(* IEC 61131-3 sources: TIA2AX/tests/test_projects/expected/HW_2200330_V18/ST30_PLC, 6 files *)

(* ---- HwInputs.st ---- *)
TYPE
	HwInputs : STRUCT
		ST30_ET200SP_CM_4xIO_Link_1 AT %B100 : ARRAY[0..31] OF BYTE;
		ST30_ET200SP_CM_4xIO_Link_2 AT %B132 : ARRAY[0..31] OF BYTE;
		ST30_ET200SP_DI_16x24VDC_ST_1 AT %B0 : WORD;
		ST30_ET200SP_DI_16x24VDC_ST_2 AT %B2 : WORD;
		ST30_ET200SP_DI_16x24VDC_ST_3 AT %B4 : WORD;
		ST30_ET200SP_DI_16x24VDC_ST_4 AT %B6 : WORD;
		ST30_ET200SP_DI_16x24VDC_ST_5 AT %B8 : WORD;
		ST30_ET200SP_DI_16x24VDC_ST_6 AT %B10 : WORD;
		ST30_1_DM260_Acquisition_Status_1 AT %B1500 : ARRAY[0..2] OF BYTE;
		ST30_1_DM260_Results_Status_1 AT %B1503 : BYTE;
		ST30_1_DM260_Soft_Event_Control_1 AT %B1504 : BYTE;
		ST30_1_DM260_Result_Data_64_bytes_1 AT %B1510 : ARRAY[0..71] OF BYTE;
		ST30_2_DM260_Acquisition_Status_1 AT %B2500 : ARRAY[0..2] OF BYTE;
		ST30_2_DM260_Results_Status_1 AT %B2503 : BYTE;
		ST30_2_DM260_Soft_Event_Control_1 AT %B2504 : BYTE;
		ST30_2_DM260_Result_Data_64_bytes_1 AT %B2510 : ARRAY[0..71] OF BYTE;
	END_STRUCT;
END_TYPE

(* ---- HwOutputs.st ---- *)
TYPE
	HwOutputs : STRUCT
		ST30_ET200SP_CM_4xIO_Link_1 AT %B100 : ARRAY[0..31] OF BYTE;
		ST30_ET200SP_CM_4xIO_Link_2 AT %B132 : ARRAY[0..31] OF BYTE;
		ST30_ET200SP_DQ_16x24VDC_0_5A_ST_1 AT %B0 : WORD;
		ST30_ET200SP_DQ_16x24VDC_0_5A_ST_2 AT %B2 : WORD;
		ST30_ET200SP_DQ_16x24VDC_0_5A_ST_3 AT %B4 : WORD;
		ST30_ET200SP_DQ_16x24VDC_0_5A_ST_4 AT %B6 : WORD;
		ST30_CPX_MPA1S_VMPA1_FB_EMS_8_8DO_1 AT %B200 : BYTE;
		ST30_CPX_MPA1G_VMPA1_FB_EMG_8_8DO_1 AT %B201 : BYTE;
		ST30_CPX_MPA1G_VMPA1_FB_EMG_8_8DO_2 AT %B202 : BYTE;
		ST30_1_DM260_Acquisition_Control_1 AT %B1500 : BYTE;
		ST30_1_DM260_Results_Control_1 AT %B1503 : BYTE;
		ST30_1_DM260_Soft_Event_Control_1 AT %B1504 : BYTE;
		ST30_1_DM260_User_Data_64_bytes_1 AT %B1510 : ARRAY[0..67] OF BYTE;
		ST30_2_DM260_Acquisition_Control_1 AT %B2500 : BYTE;
		ST30_2_DM260_Results_Control_1 AT %B2503 : BYTE;
		ST30_2_DM260_Soft_Event_Control_1 AT %B2504 : BYTE;
		ST30_2_DM260_User_Data_64_bytes_1 AT %B2510 : ARRAY[0..67] OF BYTE;
	END_STRUCT;
END_TYPE

(* ---- PlcInputs.st ---- *)
TYPE
	PlcInputs : STRUCT
		ST30_ET200SP_CM_4xIO_Link_1 : ARRAY[0..31] OF BYTE;
		ST30_ET200SP_CM_4xIO_Link_2 : ARRAY[0..31] OF BYTE;
		ST30_ET200SP_DI_16x24VDC_ST_1 : WORD;
		ST30_ET200SP_DI_16x24VDC_ST_2 : WORD;
		ST30_ET200SP_DI_16x24VDC_ST_3 : WORD;
		ST30_ET200SP_DI_16x24VDC_ST_4 : WORD;
		ST30_ET200SP_DI_16x24VDC_ST_5 : WORD;
		ST30_ET200SP_DI_16x24VDC_ST_6 : WORD;
		ST30_1_DM260_Acquisition_Status_1 : ARRAY[0..2] OF BYTE;
		ST30_1_DM260_Results_Status_1 : BYTE;
		ST30_1_DM260_Soft_Event_Control_1 : BYTE;
		ST30_1_DM260_Result_Data_64_bytes_1 : ARRAY[0..71] OF BYTE;
		ST30_2_DM260_Acquisition_Status_1 : ARRAY[0..2] OF BYTE;
		ST30_2_DM260_Results_Status_1 : BYTE;
		ST30_2_DM260_Soft_Event_Control_1 : BYTE;
		ST30_2_DM260_Result_Data_64_bytes_1 : ARRAY[0..71] OF BYTE;
	END_STRUCT;
END_TYPE

(* ---- PlcOutputs.st ---- *)
TYPE
	PlcOutputs : STRUCT
		ST30_ET200SP_CM_4xIO_Link_1 : ARRAY[0..31] OF BYTE;
		ST30_ET200SP_CM_4xIO_Link_2 : ARRAY[0..31] OF BYTE;
		ST30_ET200SP_DQ_16x24VDC_0_5A_ST_1 : WORD;
		ST30_ET200SP_DQ_16x24VDC_0_5A_ST_2 : WORD;
		ST30_ET200SP_DQ_16x24VDC_0_5A_ST_3 : WORD;
		ST30_ET200SP_DQ_16x24VDC_0_5A_ST_4 : WORD;
		ST30_CPX_MPA1S_VMPA1_FB_EMS_8_8DO_1 : BYTE;
		ST30_CPX_MPA1G_VMPA1_FB_EMG_8_8DO_1 : BYTE;
		ST30_CPX_MPA1G_VMPA1_FB_EMG_8_8DO_2 : BYTE;
		ST30_1_DM260_Acquisition_Control_1 : BYTE;
		ST30_1_DM260_Results_Control_1 : BYTE;
		ST30_1_DM260_Soft_Event_Control_1 : BYTE;
		ST30_1_DM260_User_Data_64_bytes_1 : ARRAY[0..67] OF BYTE;
		ST30_2_DM260_Acquisition_Control_1 : BYTE;
		ST30_2_DM260_Results_Control_1 : BYTE;
		ST30_2_DM260_Soft_Event_Control_1 : BYTE;
		ST30_2_DM260_User_Data_64_bytes_1 : ARRAY[0..67] OF BYTE;
	END_STRUCT;
END_TYPE

(* ---- CopyInputs.st ---- *)
FUNCTION CopyInputs
	VAR_EXTERNAL
		HwInputs : HwInputs;
		PlcInputs : PlcInputs;
	END_VAR
	PlcInputs.ST30_ET200SP_CM_4xIO_Link_1[0] := HwInputs.ST30_ET200SP_CM_4xIO_Link_1[0];
	PlcInputs.ST30_ET200SP_CM_4xIO_Link_1[1] := HwInputs.ST30_ET200SP_CM_4xIO_Link_1[1];
	PlcInputs.ST30_ET200SP_CM_4xIO_Link_1[2] := HwInputs.ST30_ET200SP_CM_4xIO_Link_1[2];
	PlcInputs.ST30_ET200SP_CM_4xIO_Link_1[3] := HwInputs.ST30_ET200SP_CM_4xIO_Link_1[3];
	PlcInputs.ST30_ET200SP_CM_4xIO_Link_1[4] := HwInputs.ST30_ET200SP_CM_4xIO_Link_1[4];
	PlcInputs.ST30_ET200SP_CM_4xIO_Link_1[5] := HwInputs.ST30_ET200SP_CM_4xIO_Link_1[5];
	PlcInputs.ST30_ET200SP_CM_4xIO_Link_1[6] := HwInputs.ST30_ET200SP_CM_4xIO_Link_1[6];
	PlcInputs.ST30_ET200SP_CM_4xIO_Link_1[7] := HwInputs.ST30_ET200SP_CM_4xIO_Link_1[7];
	PlcInputs.ST30_ET200SP_CM_4xIO_Link_1[8] := HwInputs.ST30_ET200SP_CM_4xIO_Link_1[8];
	PlcInputs.ST30_ET200SP_CM_4xIO_Link_1[9] := HwInputs.ST30_ET200SP_CM_4xIO_Link_1[9];
	PlcInputs.ST30_ET200SP_CM_4xIO_Link_1[10] := HwInputs.ST30_ET200SP_CM_4xIO_Link_1[10];
	PlcInputs.ST30_ET200SP_CM_4xIO_Link_1[11] := HwInputs.ST30_ET200SP_CM_4xIO_Link_1[11];
	PlcInputs.ST30_ET200SP_CM_4xIO_Link_1[12] := HwInputs.ST30_ET200SP_CM_4xIO_Link_1[12];
	PlcInputs.ST30_ET200SP_CM_4xIO_Link_1[13] := HwInputs.ST30_ET200SP_CM_4xIO_Link_1[13];
	PlcInputs.ST30_ET200SP_CM_4xIO_Link_1[14] := HwInputs.ST30_ET200SP_CM_4xIO_Link_1[14];
	PlcInputs.ST30_ET200SP_CM_4xIO_Link_1[15] := HwInputs.ST30_ET200SP_CM_4xIO_Link_1[15];
	PlcInputs.ST30_ET200SP_CM_4xIO_Link_1[16] := HwInputs.ST30_ET200SP_CM_4xIO_Link_1[16];
	PlcInputs.ST30_ET200SP_CM_4xIO_Link_1[17] := HwInputs.ST30_ET200SP_CM_4xIO_Link_1[17];
	PlcInputs.ST30_ET200SP_CM_4xIO_Link_1[18] := HwInputs.ST30_ET200SP_CM_4xIO_Link_1[18];
	PlcInputs.ST30_ET200SP_CM_4xIO_Link_1[19] := HwInputs.ST30_ET200SP_CM_4xIO_Link_1[19];
	PlcInputs.ST30_ET200SP_CM_4xIO_Link_1[20] := HwInputs.ST30_ET200SP_CM_4xIO_Link_1[20];
	PlcInputs.ST30_ET200SP_CM_4xIO_Link_1[21] := HwInputs.ST30_ET200SP_CM_4xIO_Link_1[21];
	PlcInputs.ST30_ET200SP_CM_4xIO_Link_1[22] := HwInputs.ST30_ET200SP_CM_4xIO_Link_1[22];
	PlcInputs.ST30_ET200SP_CM_4xIO_Link_1[23] := HwInputs.ST30_ET200SP_CM_4xIO_Link_1[23];
	PlcInputs.ST30_ET200SP_CM_4xIO_Link_1[24] := HwInputs.ST30_ET200SP_CM_4xIO_Link_1[24];
	PlcInputs.ST30_ET200SP_CM_4xIO_Link_1[25] := HwInputs.ST30_ET200SP_CM_4xIO_Link_1[25];
	PlcInputs.ST30_ET200SP_CM_4xIO_Link_1[26] := HwInputs.ST30_ET200SP_CM_4xIO_Link_1[26];
	PlcInputs.ST30_ET200SP_CM_4xIO_Link_1[27] := HwInputs.ST30_ET200SP_CM_4xIO_Link_1[27];
	PlcInputs.ST30_ET200SP_CM_4xIO_Link_1[28] := HwInputs.ST30_ET200SP_CM_4xIO_Link_1[28];
	PlcInputs.ST30_ET200SP_CM_4xIO_Link_1[29] := HwInputs.ST30_ET200SP_CM_4xIO_Link_1[29];
	PlcInputs.ST30_ET200SP_CM_4xIO_Link_1[30] := HwInputs.ST30_ET200SP_CM_4xIO_Link_1[30];
	PlcInputs.ST30_ET200SP_CM_4xIO_Link_1[31] := HwInputs.ST30_ET200SP_CM_4xIO_Link_1[31];
	PlcInputs.ST30_ET200SP_CM_4xIO_Link_2[0] := HwInputs.ST30_ET200SP_CM_4xIO_Link_2[0];
	PlcInputs.ST30_ET200SP_CM_4xIO_Link_2[1] := HwInputs.ST30_ET200SP_CM_4xIO_Link_2[1];
	PlcInputs.ST30_ET200SP_CM_4xIO_Link_2[2] := HwInputs.ST30_ET200SP_CM_4xIO_Link_2[2];
	PlcInputs.ST30_ET200SP_CM_4xIO_Link_2[3] := HwInputs.ST30_ET200SP_CM_4xIO_Link_2[3];
	PlcInputs.ST30_ET200SP_CM_4xIO_Link_2[4] := HwInputs.ST30_ET200SP_CM_4xIO_Link_2[4];
	PlcInputs.ST30_ET200SP_CM_4xIO_Link_2[5] := HwInputs.ST30_ET200SP_CM_4xIO_Link_2[5];
	PlcInputs.ST30_ET200SP_CM_4xIO_Link_2[6] := HwInputs.ST30_ET200SP_CM_4xIO_Link_2[6];
	PlcInputs.ST30_ET200SP_CM_4xIO_Link_2[7] := HwInputs.ST30_ET200SP_CM_4xIO_Link_2[7];
	PlcInputs.ST30_ET200SP_CM_4xIO_Link_2[8] := HwInputs.ST30_ET200SP_CM_4xIO_Link_2[8];
	PlcInputs.ST30_ET200SP_CM_4xIO_Link_2[9] := HwInputs.ST30_ET200SP_CM_4xIO_Link_2[9];
	PlcInputs.ST30_ET200SP_CM_4xIO_Link_2[10] := HwInputs.ST30_ET200SP_CM_4xIO_Link_2[10];
	PlcInputs.ST30_ET200SP_CM_4xIO_Link_2[11] := HwInputs.ST30_ET200SP_CM_4xIO_Link_2[11];
	PlcInputs.ST30_ET200SP_CM_4xIO_Link_2[12] := HwInputs.ST30_ET200SP_CM_4xIO_Link_2[12];
	PlcInputs.ST30_ET200SP_CM_4xIO_Link_2[13] := HwInputs.ST30_ET200SP_CM_4xIO_Link_2[13];
	PlcInputs.ST30_ET200SP_CM_4xIO_Link_2[14] := HwInputs.ST30_ET200SP_CM_4xIO_Link_2[14];
	PlcInputs.ST30_ET200SP_CM_4xIO_Link_2[15] := HwInputs.ST30_ET200SP_CM_4xIO_Link_2[15];
	PlcInputs.ST30_ET200SP_CM_4xIO_Link_2[16] := HwInputs.ST30_ET200SP_CM_4xIO_Link_2[16];
	PlcInputs.ST30_ET200SP_CM_4xIO_Link_2[17] := HwInputs.ST30_ET200SP_CM_4xIO_Link_2[17];
	PlcInputs.ST30_ET200SP_CM_4xIO_Link_2[18] := HwInputs.ST30_ET200SP_CM_4xIO_Link_2[18];
	PlcInputs.ST30_ET200SP_CM_4xIO_Link_2[19] := HwInputs.ST30_ET200SP_CM_4xIO_Link_2[19];
	PlcInputs.ST30_ET200SP_CM_4xIO_Link_2[20] := HwInputs.ST30_ET200SP_CM_4xIO_Link_2[20];
	PlcInputs.ST30_ET200SP_CM_4xIO_Link_2[21] := HwInputs.ST30_ET200SP_CM_4xIO_Link_2[21];
	PlcInputs.ST30_ET200SP_CM_4xIO_Link_2[22] := HwInputs.ST30_ET200SP_CM_4xIO_Link_2[22];
	PlcInputs.ST30_ET200SP_CM_4xIO_Link_2[23] := HwInputs.ST30_ET200SP_CM_4xIO_Link_2[23];
	PlcInputs.ST30_ET200SP_CM_4xIO_Link_2[24] := HwInputs.ST30_ET200SP_CM_4xIO_Link_2[24];
	PlcInputs.ST30_ET200SP_CM_4xIO_Link_2[25] := HwInputs.ST30_ET200SP_CM_4xIO_Link_2[25];
	PlcInputs.ST30_ET200SP_CM_4xIO_Link_2[26] := HwInputs.ST30_ET200SP_CM_4xIO_Link_2[26];
	PlcInputs.ST30_ET200SP_CM_4xIO_Link_2[27] := HwInputs.ST30_ET200SP_CM_4xIO_Link_2[27];
	PlcInputs.ST30_ET200SP_CM_4xIO_Link_2[28] := HwInputs.ST30_ET200SP_CM_4xIO_Link_2[28];
	PlcInputs.ST30_ET200SP_CM_4xIO_Link_2[29] := HwInputs.ST30_ET200SP_CM_4xIO_Link_2[29];
	PlcInputs.ST30_ET200SP_CM_4xIO_Link_2[30] := HwInputs.ST30_ET200SP_CM_4xIO_Link_2[30];
	PlcInputs.ST30_ET200SP_CM_4xIO_Link_2[31] := HwInputs.ST30_ET200SP_CM_4xIO_Link_2[31];
	PlcInputs.ST30_ET200SP_DI_16x24VDC_ST_1 := HwInputs.ST30_ET200SP_DI_16x24VDC_ST_1;
	PlcInputs.ST30_ET200SP_DI_16x24VDC_ST_2 := HwInputs.ST30_ET200SP_DI_16x24VDC_ST_2;
	PlcInputs.ST30_ET200SP_DI_16x24VDC_ST_3 := HwInputs.ST30_ET200SP_DI_16x24VDC_ST_3;
	PlcInputs.ST30_ET200SP_DI_16x24VDC_ST_4 := HwInputs.ST30_ET200SP_DI_16x24VDC_ST_4;
	PlcInputs.ST30_ET200SP_DI_16x24VDC_ST_5 := HwInputs.ST30_ET200SP_DI_16x24VDC_ST_5;
	PlcInputs.ST30_ET200SP_DI_16x24VDC_ST_6 := HwInputs.ST30_ET200SP_DI_16x24VDC_ST_6;
	PlcInputs.ST30_1_DM260_Acquisition_Status_1[0] := HwInputs.ST30_1_DM260_Acquisition_Status_1[0];
	PlcInputs.ST30_1_DM260_Acquisition_Status_1[1] := HwInputs.ST30_1_DM260_Acquisition_Status_1[1];
	PlcInputs.ST30_1_DM260_Acquisition_Status_1[2] := HwInputs.ST30_1_DM260_Acquisition_Status_1[2];
	PlcInputs.ST30_1_DM260_Results_Status_1 := HwInputs.ST30_1_DM260_Results_Status_1;
	PlcInputs.ST30_1_DM260_Soft_Event_Control_1 := HwInputs.ST30_1_DM260_Soft_Event_Control_1;
	PlcInputs.ST30_1_DM260_Result_Data_64_bytes_1[0] := HwInputs.ST30_1_DM260_Result_Data_64_bytes_1[0];
	PlcInputs.ST30_1_DM260_Result_Data_64_bytes_1[1] := HwInputs.ST30_1_DM260_Result_Data_64_bytes_1[1];
	PlcInputs.ST30_1_DM260_Result_Data_64_bytes_1[2] := HwInputs.ST30_1_DM260_Result_Data_64_bytes_1[2];
	PlcInputs.ST30_1_DM260_Result_Data_64_bytes_1[3] := HwInputs.ST30_1_DM260_Result_Data_64_bytes_1[3];
	PlcInputs.ST30_1_DM260_Result_Data_64_bytes_1[4] := HwInputs.ST30_1_DM260_Result_Data_64_bytes_1[4];
	PlcInputs.ST30_1_DM260_Result_Data_64_bytes_1[5] := HwInputs.ST30_1_DM260_Result_Data_64_bytes_1[5];
	PlcInputs.ST30_1_DM260_Result_Data_64_bytes_1[6] := HwInputs.ST30_1_DM260_Result_Data_64_bytes_1[6];
	PlcInputs.ST30_1_DM260_Result_Data_64_bytes_1[7] := HwInputs.ST30_1_DM260_Result_Data_64_bytes_1[7];
	PlcInputs.ST30_1_DM260_Result_Data_64_bytes_1[8] := HwInputs.ST30_1_DM260_Result_Data_64_bytes_1[8];
	PlcInputs.ST30_1_DM260_Result_Data_64_bytes_1[9] := HwInputs.ST30_1_DM260_Result_Data_64_bytes_1[9];
	PlcInputs.ST30_1_DM260_Result_Data_64_bytes_1[10] := HwInputs.ST30_1_DM260_Result_Data_64_bytes_1[10];
	PlcInputs.ST30_1_DM260_Result_Data_64_bytes_1[11] := HwInputs.ST30_1_DM260_Result_Data_64_bytes_1[11];
	PlcInputs.ST30_1_DM260_Result_Data_64_bytes_1[12] := HwInputs.ST30_1_DM260_Result_Data_64_bytes_1[12];
	PlcInputs.ST30_1_DM260_Result_Data_64_bytes_1[13] := HwInputs.ST30_1_DM260_Result_Data_64_bytes_1[13];
	PlcInputs.ST30_1_DM260_Result_Data_64_bytes_1[14] := HwInputs.ST30_1_DM260_Result_Data_64_bytes_1[14];
	PlcInputs.ST30_1_DM260_Result_Data_64_bytes_1[15] := HwInputs.ST30_1_DM260_Result_Data_64_bytes_1[15];
	PlcInputs.ST30_1_DM260_Result_Data_64_bytes_1[16] := HwInputs.ST30_1_DM260_Result_Data_64_bytes_1[16];
	PlcInputs.ST30_1_DM260_Result_Data_64_bytes_1[17] := HwInputs.ST30_1_DM260_Result_Data_64_bytes_1[17];
	PlcInputs.ST30_1_DM260_Result_Data_64_bytes_1[18] := HwInputs.ST30_1_DM260_Result_Data_64_bytes_1[18];
	PlcInputs.ST30_1_DM260_Result_Data_64_bytes_1[19] := HwInputs.ST30_1_DM260_Result_Data_64_bytes_1[19];
	PlcInputs.ST30_1_DM260_Result_Data_64_bytes_1[20] := HwInputs.ST30_1_DM260_Result_Data_64_bytes_1[20];
	PlcInputs.ST30_1_DM260_Result_Data_64_bytes_1[21] := HwInputs.ST30_1_DM260_Result_Data_64_bytes_1[21];
	PlcInputs.ST30_1_DM260_Result_Data_64_bytes_1[22] := HwInputs.ST30_1_DM260_Result_Data_64_bytes_1[22];
	PlcInputs.ST30_1_DM260_Result_Data_64_bytes_1[23] := HwInputs.ST30_1_DM260_Result_Data_64_bytes_1[23];
	PlcInputs.ST30_1_DM260_Result_Data_64_bytes_1[24] := HwInputs.ST30_1_DM260_Result_Data_64_bytes_1[24];
	PlcInputs.ST30_1_DM260_Result_Data_64_bytes_1[25] := HwInputs.ST30_1_DM260_Result_Data_64_bytes_1[25];
	PlcInputs.ST30_1_DM260_Result_Data_64_bytes_1[26] := HwInputs.ST30_1_DM260_Result_Data_64_bytes_1[26];
	PlcInputs.ST30_1_DM260_Result_Data_64_bytes_1[27] := HwInputs.ST30_1_DM260_Result_Data_64_bytes_1[27];
	PlcInputs.ST30_1_DM260_Result_Data_64_bytes_1[28] := HwInputs.ST30_1_DM260_Result_Data_64_bytes_1[28];
	PlcInputs.ST30_1_DM260_Result_Data_64_bytes_1[29] := HwInputs.ST30_1_DM260_Result_Data_64_bytes_1[29];
	PlcInputs.ST30_1_DM260_Result_Data_64_bytes_1[30] := HwInputs.ST30_1_DM260_Result_Data_64_bytes_1[30];
	PlcInputs.ST30_1_DM260_Result_Data_64_bytes_1[31] := HwInputs.ST30_1_DM260_Result_Data_64_bytes_1[31];
	PlcInputs.ST30_1_DM260_Result_Data_64_bytes_1[32] := HwInputs.ST30_1_DM260_Result_Data_64_bytes_1[32];
	PlcInputs.ST30_1_DM260_Result_Data_64_bytes_1[33] := HwInputs.ST30_1_DM260_Result_Data_64_bytes_1[33];
	PlcInputs.ST30_1_DM260_Result_Data_64_bytes_1[34] := HwInputs.ST30_1_DM260_Result_Data_64_bytes_1[34];
	PlcInputs.ST30_1_DM260_Result_Data_64_bytes_1[35] := HwInputs.ST30_1_DM260_Result_Data_64_bytes_1[35];
	PlcInputs.ST30_1_DM260_Result_Data_64_bytes_1[36] := HwInputs.ST30_1_DM260_Result_Data_64_bytes_1[36];
	PlcInputs.ST30_1_DM260_Result_Data_64_bytes_1[37] := HwInputs.ST30_1_DM260_Result_Data_64_bytes_1[37];
	PlcInputs.ST30_1_DM260_Result_Data_64_bytes_1[38] := HwInputs.ST30_1_DM260_Result_Data_64_bytes_1[38];
	PlcInputs.ST30_1_DM260_Result_Data_64_bytes_1[39] := HwInputs.ST30_1_DM260_Result_Data_64_bytes_1[39];
	PlcInputs.ST30_1_DM260_Result_Data_64_bytes_1[40] := HwInputs.ST30_1_DM260_Result_Data_64_bytes_1[40];
	PlcInputs.ST30_1_DM260_Result_Data_64_bytes_1[41] := HwInputs.ST30_1_DM260_Result_Data_64_bytes_1[41];
	PlcInputs.ST30_1_DM260_Result_Data_64_bytes_1[42] := HwInputs.ST30_1_DM260_Result_Data_64_bytes_1[42];
	PlcInputs.ST30_1_DM260_Result_Data_64_bytes_1[43] := HwInputs.ST30_1_DM260_Result_Data_64_bytes_1[43];
	PlcInputs.ST30_1_DM260_Result_Data_64_bytes_1[44] := HwInputs.ST30_1_DM260_Result_Data_64_bytes_1[44];
	PlcInputs.ST30_1_DM260_Result_Data_64_bytes_1[45] := HwInputs.ST30_1_DM260_Result_Data_64_bytes_1[45];
	PlcInputs.ST30_1_DM260_Result_Data_64_bytes_1[46] := HwInputs.ST30_1_DM260_Result_Data_64_bytes_1[46];
	PlcInputs.ST30_1_DM260_Result_Data_64_bytes_1[47] := HwInputs.ST30_1_DM260_Result_Data_64_bytes_1[47];
	PlcInputs.ST30_1_DM260_Result_Data_64_bytes_1[48] := HwInputs.ST30_1_DM260_Result_Data_64_bytes_1[48];
	PlcInputs.ST30_1_DM260_Result_Data_64_bytes_1[49] := HwInputs.ST30_1_DM260_Result_Data_64_bytes_1[49];
	PlcInputs.ST30_1_DM260_Result_Data_64_bytes_1[50] := HwInputs.ST30_1_DM260_Result_Data_64_bytes_1[50];
	PlcInputs.ST30_1_DM260_Result_Data_64_bytes_1[51] := HwInputs.ST30_1_DM260_Result_Data_64_bytes_1[51];
	PlcInputs.ST30_1_DM260_Result_Data_64_bytes_1[52] := HwInputs.ST30_1_DM260_Result_Data_64_bytes_1[52];
	PlcInputs.ST30_1_DM260_Result_Data_64_bytes_1[53] := HwInputs.ST30_1_DM260_Result_Data_64_bytes_1[53];
	PlcInputs.ST30_1_DM260_Result_Data_64_bytes_1[54] := HwInputs.ST30_1_DM260_Result_Data_64_bytes_1[54];
	PlcInputs.ST30_1_DM260_Result_Data_64_bytes_1[55] := HwInputs.ST30_1_DM260_Result_Data_64_bytes_1[55];
	PlcInputs.ST30_1_DM260_Result_Data_64_bytes_1[56] := HwInputs.ST30_1_DM260_Result_Data_64_bytes_1[56];
	PlcInputs.ST30_1_DM260_Result_Data_64_bytes_1[57] := HwInputs.ST30_1_DM260_Result_Data_64_bytes_1[57];
	PlcInputs.ST30_1_DM260_Result_Data_64_bytes_1[58] := HwInputs.ST30_1_DM260_Result_Data_64_bytes_1[58];
	PlcInputs.ST30_1_DM260_Result_Data_64_bytes_1[59] := HwInputs.ST30_1_DM260_Result_Data_64_bytes_1[59];
	PlcInputs.ST30_1_DM260_Result_Data_64_bytes_1[60] := HwInputs.ST30_1_DM260_Result_Data_64_bytes_1[60];
	PlcInputs.ST30_1_DM260_Result_Data_64_bytes_1[61] := HwInputs.ST30_1_DM260_Result_Data_64_bytes_1[61];
	PlcInputs.ST30_1_DM260_Result_Data_64_bytes_1[62] := HwInputs.ST30_1_DM260_Result_Data_64_bytes_1[62];
	PlcInputs.ST30_1_DM260_Result_Data_64_bytes_1[63] := HwInputs.ST30_1_DM260_Result_Data_64_bytes_1[63];
	PlcInputs.ST30_1_DM260_Result_Data_64_bytes_1[64] := HwInputs.ST30_1_DM260_Result_Data_64_bytes_1[64];
	PlcInputs.ST30_1_DM260_Result_Data_64_bytes_1[65] := HwInputs.ST30_1_DM260_Result_Data_64_bytes_1[65];
	PlcInputs.ST30_1_DM260_Result_Data_64_bytes_1[66] := HwInputs.ST30_1_DM260_Result_Data_64_bytes_1[66];
	PlcInputs.ST30_1_DM260_Result_Data_64_bytes_1[67] := HwInputs.ST30_1_DM260_Result_Data_64_bytes_1[67];
	PlcInputs.ST30_1_DM260_Result_Data_64_bytes_1[68] := HwInputs.ST30_1_DM260_Result_Data_64_bytes_1[68];
	PlcInputs.ST30_1_DM260_Result_Data_64_bytes_1[69] := HwInputs.ST30_1_DM260_Result_Data_64_bytes_1[69];
	PlcInputs.ST30_1_DM260_Result_Data_64_bytes_1[70] := HwInputs.ST30_1_DM260_Result_Data_64_bytes_1[70];
	PlcInputs.ST30_1_DM260_Result_Data_64_bytes_1[71] := HwInputs.ST30_1_DM260_Result_Data_64_bytes_1[71];
	PlcInputs.ST30_2_DM260_Acquisition_Status_1[0] := HwInputs.ST30_2_DM260_Acquisition_Status_1[0];
	PlcInputs.ST30_2_DM260_Acquisition_Status_1[1] := HwInputs.ST30_2_DM260_Acquisition_Status_1[1];
	PlcInputs.ST30_2_DM260_Acquisition_Status_1[2] := HwInputs.ST30_2_DM260_Acquisition_Status_1[2];
	PlcInputs.ST30_2_DM260_Results_Status_1 := HwInputs.ST30_2_DM260_Results_Status_1;
	PlcInputs.ST30_2_DM260_Soft_Event_Control_1 := HwInputs.ST30_2_DM260_Soft_Event_Control_1;
	PlcInputs.ST30_2_DM260_Result_Data_64_bytes_1[0] := HwInputs.ST30_2_DM260_Result_Data_64_bytes_1[0];
	PlcInputs.ST30_2_DM260_Result_Data_64_bytes_1[1] := HwInputs.ST30_2_DM260_Result_Data_64_bytes_1[1];
	PlcInputs.ST30_2_DM260_Result_Data_64_bytes_1[2] := HwInputs.ST30_2_DM260_Result_Data_64_bytes_1[2];
	PlcInputs.ST30_2_DM260_Result_Data_64_bytes_1[3] := HwInputs.ST30_2_DM260_Result_Data_64_bytes_1[3];
	PlcInputs.ST30_2_DM260_Result_Data_64_bytes_1[4] := HwInputs.ST30_2_DM260_Result_Data_64_bytes_1[4];
	PlcInputs.ST30_2_DM260_Result_Data_64_bytes_1[5] := HwInputs.ST30_2_DM260_Result_Data_64_bytes_1[5];
	PlcInputs.ST30_2_DM260_Result_Data_64_bytes_1[6] := HwInputs.ST30_2_DM260_Result_Data_64_bytes_1[6];
	PlcInputs.ST30_2_DM260_Result_Data_64_bytes_1[7] := HwInputs.ST30_2_DM260_Result_Data_64_bytes_1[7];
	PlcInputs.ST30_2_DM260_Result_Data_64_bytes_1[8] := HwInputs.ST30_2_DM260_Result_Data_64_bytes_1[8];
	PlcInputs.ST30_2_DM260_Result_Data_64_bytes_1[9] := HwInputs.ST30_2_DM260_Result_Data_64_bytes_1[9];
	PlcInputs.ST30_2_DM260_Result_Data_64_bytes_1[10] := HwInputs.ST30_2_DM260_Result_Data_64_bytes_1[10];
	PlcInputs.ST30_2_DM260_Result_Data_64_bytes_1[11] := HwInputs.ST30_2_DM260_Result_Data_64_bytes_1[11];
	PlcInputs.ST30_2_DM260_Result_Data_64_bytes_1[12] := HwInputs.ST30_2_DM260_Result_Data_64_bytes_1[12];
	PlcInputs.ST30_2_DM260_Result_Data_64_bytes_1[13] := HwInputs.ST30_2_DM260_Result_Data_64_bytes_1[13];
	PlcInputs.ST30_2_DM260_Result_Data_64_bytes_1[14] := HwInputs.ST30_2_DM260_Result_Data_64_bytes_1[14];
	PlcInputs.ST30_2_DM260_Result_Data_64_bytes_1[15] := HwInputs.ST30_2_DM260_Result_Data_64_bytes_1[15];
	PlcInputs.ST30_2_DM260_Result_Data_64_bytes_1[16] := HwInputs.ST30_2_DM260_Result_Data_64_bytes_1[16];
	PlcInputs.ST30_2_DM260_Result_Data_64_bytes_1[17] := HwInputs.ST30_2_DM260_Result_Data_64_bytes_1[17];
	PlcInputs.ST30_2_DM260_Result_Data_64_bytes_1[18] := HwInputs.ST30_2_DM260_Result_Data_64_bytes_1[18];
	PlcInputs.ST30_2_DM260_Result_Data_64_bytes_1[19] := HwInputs.ST30_2_DM260_Result_Data_64_bytes_1[19];
	PlcInputs.ST30_2_DM260_Result_Data_64_bytes_1[20] := HwInputs.ST30_2_DM260_Result_Data_64_bytes_1[20];
	PlcInputs.ST30_2_DM260_Result_Data_64_bytes_1[21] := HwInputs.ST30_2_DM260_Result_Data_64_bytes_1[21];
	PlcInputs.ST30_2_DM260_Result_Data_64_bytes_1[22] := HwInputs.ST30_2_DM260_Result_Data_64_bytes_1[22];
	PlcInputs.ST30_2_DM260_Result_Data_64_bytes_1[23] := HwInputs.ST30_2_DM260_Result_Data_64_bytes_1[23];
	PlcInputs.ST30_2_DM260_Result_Data_64_bytes_1[24] := HwInputs.ST30_2_DM260_Result_Data_64_bytes_1[24];
	PlcInputs.ST30_2_DM260_Result_Data_64_bytes_1[25] := HwInputs.ST30_2_DM260_Result_Data_64_bytes_1[25];
	PlcInputs.ST30_2_DM260_Result_Data_64_bytes_1[26] := HwInputs.ST30_2_DM260_Result_Data_64_bytes_1[26];
	PlcInputs.ST30_2_DM260_Result_Data_64_bytes_1[27] := HwInputs.ST30_2_DM260_Result_Data_64_bytes_1[27];
	PlcInputs.ST30_2_DM260_Result_Data_64_bytes_1[28] := HwInputs.ST30_2_DM260_Result_Data_64_bytes_1[28];
	PlcInputs.ST30_2_DM260_Result_Data_64_bytes_1[29] := HwInputs.ST30_2_DM260_Result_Data_64_bytes_1[29];
	PlcInputs.ST30_2_DM260_Result_Data_64_bytes_1[30] := HwInputs.ST30_2_DM260_Result_Data_64_bytes_1[30];
	PlcInputs.ST30_2_DM260_Result_Data_64_bytes_1[31] := HwInputs.ST30_2_DM260_Result_Data_64_bytes_1[31];
	PlcInputs.ST30_2_DM260_Result_Data_64_bytes_1[32] := HwInputs.ST30_2_DM260_Result_Data_64_bytes_1[32];
	PlcInputs.ST30_2_DM260_Result_Data_64_bytes_1[33] := HwInputs.ST30_2_DM260_Result_Data_64_bytes_1[33];
	PlcInputs.ST30_2_DM260_Result_Data_64_bytes_1[34] := HwInputs.ST30_2_DM260_Result_Data_64_bytes_1[34];
	PlcInputs.ST30_2_DM260_Result_Data_64_bytes_1[35] := HwInputs.ST30_2_DM260_Result_Data_64_bytes_1[35];
	PlcInputs.ST30_2_DM260_Result_Data_64_bytes_1[36] := HwInputs.ST30_2_DM260_Result_Data_64_bytes_1[36];
	PlcInputs.ST30_2_DM260_Result_Data_64_bytes_1[37] := HwInputs.ST30_2_DM260_Result_Data_64_bytes_1[37];
	PlcInputs.ST30_2_DM260_Result_Data_64_bytes_1[38] := HwInputs.ST30_2_DM260_Result_Data_64_bytes_1[38];
	PlcInputs.ST30_2_DM260_Result_Data_64_bytes_1[39] := HwInputs.ST30_2_DM260_Result_Data_64_bytes_1[39];
	PlcInputs.ST30_2_DM260_Result_Data_64_bytes_1[40] := HwInputs.ST30_2_DM260_Result_Data_64_bytes_1[40];
	PlcInputs.ST30_2_DM260_Result_Data_64_bytes_1[41] := HwInputs.ST30_2_DM260_Result_Data_64_bytes_1[41];
	PlcInputs.ST30_2_DM260_Result_Data_64_bytes_1[42] := HwInputs.ST30_2_DM260_Result_Data_64_bytes_1[42];
	PlcInputs.ST30_2_DM260_Result_Data_64_bytes_1[43] := HwInputs.ST30_2_DM260_Result_Data_64_bytes_1[43];
	PlcInputs.ST30_2_DM260_Result_Data_64_bytes_1[44] := HwInputs.ST30_2_DM260_Result_Data_64_bytes_1[44];
	PlcInputs.ST30_2_DM260_Result_Data_64_bytes_1[45] := HwInputs.ST30_2_DM260_Result_Data_64_bytes_1[45];
	PlcInputs.ST30_2_DM260_Result_Data_64_bytes_1[46] := HwInputs.ST30_2_DM260_Result_Data_64_bytes_1[46];
	PlcInputs.ST30_2_DM260_Result_Data_64_bytes_1[47] := HwInputs.ST30_2_DM260_Result_Data_64_bytes_1[47];
	PlcInputs.ST30_2_DM260_Result_Data_64_bytes_1[48] := HwInputs.ST30_2_DM260_Result_Data_64_bytes_1[48];
	PlcInputs.ST30_2_DM260_Result_Data_64_bytes_1[49] := HwInputs.ST30_2_DM260_Result_Data_64_bytes_1[49];
	PlcInputs.ST30_2_DM260_Result_Data_64_bytes_1[50] := HwInputs.ST30_2_DM260_Result_Data_64_bytes_1[50];
	PlcInputs.ST30_2_DM260_Result_Data_64_bytes_1[51] := HwInputs.ST30_2_DM260_Result_Data_64_bytes_1[51];
	PlcInputs.ST30_2_DM260_Result_Data_64_bytes_1[52] := HwInputs.ST30_2_DM260_Result_Data_64_bytes_1[52];
	PlcInputs.ST30_2_DM260_Result_Data_64_bytes_1[53] := HwInputs.ST30_2_DM260_Result_Data_64_bytes_1[53];
	PlcInputs.ST30_2_DM260_Result_Data_64_bytes_1[54] := HwInputs.ST30_2_DM260_Result_Data_64_bytes_1[54];
	PlcInputs.ST30_2_DM260_Result_Data_64_bytes_1[55] := HwInputs.ST30_2_DM260_Result_Data_64_bytes_1[55];
	PlcInputs.ST30_2_DM260_Result_Data_64_bytes_1[56] := HwInputs.ST30_2_DM260_Result_Data_64_bytes_1[56];
	PlcInputs.ST30_2_DM260_Result_Data_64_bytes_1[57] := HwInputs.ST30_2_DM260_Result_Data_64_bytes_1[57];
	PlcInputs.ST30_2_DM260_Result_Data_64_bytes_1[58] := HwInputs.ST30_2_DM260_Result_Data_64_bytes_1[58];
	PlcInputs.ST30_2_DM260_Result_Data_64_bytes_1[59] := HwInputs.ST30_2_DM260_Result_Data_64_bytes_1[59];
	PlcInputs.ST30_2_DM260_Result_Data_64_bytes_1[60] := HwInputs.ST30_2_DM260_Result_Data_64_bytes_1[60];
	PlcInputs.ST30_2_DM260_Result_Data_64_bytes_1[61] := HwInputs.ST30_2_DM260_Result_Data_64_bytes_1[61];
	PlcInputs.ST30_2_DM260_Result_Data_64_bytes_1[62] := HwInputs.ST30_2_DM260_Result_Data_64_bytes_1[62];
	PlcInputs.ST30_2_DM260_Result_Data_64_bytes_1[63] := HwInputs.ST30_2_DM260_Result_Data_64_bytes_1[63];
	PlcInputs.ST30_2_DM260_Result_Data_64_bytes_1[64] := HwInputs.ST30_2_DM260_Result_Data_64_bytes_1[64];
	PlcInputs.ST30_2_DM260_Result_Data_64_bytes_1[65] := HwInputs.ST30_2_DM260_Result_Data_64_bytes_1[65];
	PlcInputs.ST30_2_DM260_Result_Data_64_bytes_1[66] := HwInputs.ST30_2_DM260_Result_Data_64_bytes_1[66];
	PlcInputs.ST30_2_DM260_Result_Data_64_bytes_1[67] := HwInputs.ST30_2_DM260_Result_Data_64_bytes_1[67];
	PlcInputs.ST30_2_DM260_Result_Data_64_bytes_1[68] := HwInputs.ST30_2_DM260_Result_Data_64_bytes_1[68];
	PlcInputs.ST30_2_DM260_Result_Data_64_bytes_1[69] := HwInputs.ST30_2_DM260_Result_Data_64_bytes_1[69];
	PlcInputs.ST30_2_DM260_Result_Data_64_bytes_1[70] := HwInputs.ST30_2_DM260_Result_Data_64_bytes_1[70];
	PlcInputs.ST30_2_DM260_Result_Data_64_bytes_1[71] := HwInputs.ST30_2_DM260_Result_Data_64_bytes_1[71];
END_FUNCTION

(* ---- CopyOutputs.st ---- *)
FUNCTION CopyOutputs
	VAR_EXTERNAL
		HwOutputs : HwOutputs;
		PlcOutputs : PlcOutputs;
	END_VAR
	HwOutputs.ST30_ET200SP_CM_4xIO_Link_1[0] := PlcOutputs.ST30_ET200SP_CM_4xIO_Link_1[0];
	HwOutputs.ST30_ET200SP_CM_4xIO_Link_1[1] := PlcOutputs.ST30_ET200SP_CM_4xIO_Link_1[1];
	HwOutputs.ST30_ET200SP_CM_4xIO_Link_1[2] := PlcOutputs.ST30_ET200SP_CM_4xIO_Link_1[2];
	HwOutputs.ST30_ET200SP_CM_4xIO_Link_1[3] := PlcOutputs.ST30_ET200SP_CM_4xIO_Link_1[3];
	HwOutputs.ST30_ET200SP_CM_4xIO_Link_1[4] := PlcOutputs.ST30_ET200SP_CM_4xIO_Link_1[4];
	HwOutputs.ST30_ET200SP_CM_4xIO_Link_1[5] := PlcOutputs.ST30_ET200SP_CM_4xIO_Link_1[5];
	HwOutputs.ST30_ET200SP_CM_4xIO_Link_1[6] := PlcOutputs.ST30_ET200SP_CM_4xIO_Link_1[6];
	HwOutputs.ST30_ET200SP_CM_4xIO_Link_1[7] := PlcOutputs.ST30_ET200SP_CM_4xIO_Link_1[7];
	HwOutputs.ST30_ET200SP_CM_4xIO_Link_1[8] := PlcOutputs.ST30_ET200SP_CM_4xIO_Link_1[8];
	HwOutputs.ST30_ET200SP_CM_4xIO_Link_1[9] := PlcOutputs.ST30_ET200SP_CM_4xIO_Link_1[9];
	HwOutputs.ST30_ET200SP_CM_4xIO_Link_1[10] := PlcOutputs.ST30_ET200SP_CM_4xIO_Link_1[10];
	HwOutputs.ST30_ET200SP_CM_4xIO_Link_1[11] := PlcOutputs.ST30_ET200SP_CM_4xIO_Link_1[11];
	HwOutputs.ST30_ET200SP_CM_4xIO_Link_1[12] := PlcOutputs.ST30_ET200SP_CM_4xIO_Link_1[12];
	HwOutputs.ST30_ET200SP_CM_4xIO_Link_1[13] := PlcOutputs.ST30_ET200SP_CM_4xIO_Link_1[13];
	HwOutputs.ST30_ET200SP_CM_4xIO_Link_1[14] := PlcOutputs.ST30_ET200SP_CM_4xIO_Link_1[14];
	HwOutputs.ST30_ET200SP_CM_4xIO_Link_1[15] := PlcOutputs.ST30_ET200SP_CM_4xIO_Link_1[15];
	HwOutputs.ST30_ET200SP_CM_4xIO_Link_1[16] := PlcOutputs.ST30_ET200SP_CM_4xIO_Link_1[16];
	HwOutputs.ST30_ET200SP_CM_4xIO_Link_1[17] := PlcOutputs.ST30_ET200SP_CM_4xIO_Link_1[17];
	HwOutputs.ST30_ET200SP_CM_4xIO_Link_1[18] := PlcOutputs.ST30_ET200SP_CM_4xIO_Link_1[18];
	HwOutputs.ST30_ET200SP_CM_4xIO_Link_1[19] := PlcOutputs.ST30_ET200SP_CM_4xIO_Link_1[19];
	HwOutputs.ST30_ET200SP_CM_4xIO_Link_1[20] := PlcOutputs.ST30_ET200SP_CM_4xIO_Link_1[20];
	HwOutputs.ST30_ET200SP_CM_4xIO_Link_1[21] := PlcOutputs.ST30_ET200SP_CM_4xIO_Link_1[21];
	HwOutputs.ST30_ET200SP_CM_4xIO_Link_1[22] := PlcOutputs.ST30_ET200SP_CM_4xIO_Link_1[22];
	HwOutputs.ST30_ET200SP_CM_4xIO_Link_1[23] := PlcOutputs.ST30_ET200SP_CM_4xIO_Link_1[23];
	HwOutputs.ST30_ET200SP_CM_4xIO_Link_1[24] := PlcOutputs.ST30_ET200SP_CM_4xIO_Link_1[24];
	HwOutputs.ST30_ET200SP_CM_4xIO_Link_1[25] := PlcOutputs.ST30_ET200SP_CM_4xIO_Link_1[25];
	HwOutputs.ST30_ET200SP_CM_4xIO_Link_1[26] := PlcOutputs.ST30_ET200SP_CM_4xIO_Link_1[26];
	HwOutputs.ST30_ET200SP_CM_4xIO_Link_1[27] := PlcOutputs.ST30_ET200SP_CM_4xIO_Link_1[27];
	HwOutputs.ST30_ET200SP_CM_4xIO_Link_1[28] := PlcOutputs.ST30_ET200SP_CM_4xIO_Link_1[28];
	HwOutputs.ST30_ET200SP_CM_4xIO_Link_1[29] := PlcOutputs.ST30_ET200SP_CM_4xIO_Link_1[29];
	HwOutputs.ST30_ET200SP_CM_4xIO_Link_1[30] := PlcOutputs.ST30_ET200SP_CM_4xIO_Link_1[30];
	HwOutputs.ST30_ET200SP_CM_4xIO_Link_1[31] := PlcOutputs.ST30_ET200SP_CM_4xIO_Link_1[31];
	HwOutputs.ST30_ET200SP_CM_4xIO_Link_2[0] := PlcOutputs.ST30_ET200SP_CM_4xIO_Link_2[0];
	HwOutputs.ST30_ET200SP_CM_4xIO_Link_2[1] := PlcOutputs.ST30_ET200SP_CM_4xIO_Link_2[1];
	HwOutputs.ST30_ET200SP_CM_4xIO_Link_2[2] := PlcOutputs.ST30_ET200SP_CM_4xIO_Link_2[2];
	HwOutputs.ST30_ET200SP_CM_4xIO_Link_2[3] := PlcOutputs.ST30_ET200SP_CM_4xIO_Link_2[3];
	HwOutputs.ST30_ET200SP_CM_4xIO_Link_2[4] := PlcOutputs.ST30_ET200SP_CM_4xIO_Link_2[4];
	HwOutputs.ST30_ET200SP_CM_4xIO_Link_2[5] := PlcOutputs.ST30_ET200SP_CM_4xIO_Link_2[5];
	HwOutputs.ST30_ET200SP_CM_4xIO_Link_2[6] := PlcOutputs.ST30_ET200SP_CM_4xIO_Link_2[6];
	HwOutputs.ST30_ET200SP_CM_4xIO_Link_2[7] := PlcOutputs.ST30_ET200SP_CM_4xIO_Link_2[7];
	HwOutputs.ST30_ET200SP_CM_4xIO_Link_2[8] := PlcOutputs.ST30_ET200SP_CM_4xIO_Link_2[8];
	HwOutputs.ST30_ET200SP_CM_4xIO_Link_2[9] := PlcOutputs.ST30_ET200SP_CM_4xIO_Link_2[9];
	HwOutputs.ST30_ET200SP_CM_4xIO_Link_2[10] := PlcOutputs.ST30_ET200SP_CM_4xIO_Link_2[10];
	HwOutputs.ST30_ET200SP_CM_4xIO_Link_2[11] := PlcOutputs.ST30_ET200SP_CM_4xIO_Link_2[11];
	HwOutputs.ST30_ET200SP_CM_4xIO_Link_2[12] := PlcOutputs.ST30_ET200SP_CM_4xIO_Link_2[12];
	HwOutputs.ST30_ET200SP_CM_4xIO_Link_2[13] := PlcOutputs.ST30_ET200SP_CM_4xIO_Link_2[13];
	HwOutputs.ST30_ET200SP_CM_4xIO_Link_2[14] := PlcOutputs.ST30_ET200SP_CM_4xIO_Link_2[14];
	HwOutputs.ST30_ET200SP_CM_4xIO_Link_2[15] := PlcOutputs.ST30_ET200SP_CM_4xIO_Link_2[15];
	HwOutputs.ST30_ET200SP_CM_4xIO_Link_2[16] := PlcOutputs.ST30_ET200SP_CM_4xIO_Link_2[16];
	HwOutputs.ST30_ET200SP_CM_4xIO_Link_2[17] := PlcOutputs.ST30_ET200SP_CM_4xIO_Link_2[17];
	HwOutputs.ST30_ET200SP_CM_4xIO_Link_2[18] := PlcOutputs.ST30_ET200SP_CM_4xIO_Link_2[18];
	HwOutputs.ST30_ET200SP_CM_4xIO_Link_2[19] := PlcOutputs.ST30_ET200SP_CM_4xIO_Link_2[19];
	HwOutputs.ST30_ET200SP_CM_4xIO_Link_2[20] := PlcOutputs.ST30_ET200SP_CM_4xIO_Link_2[20];
	HwOutputs.ST30_ET200SP_CM_4xIO_Link_2[21] := PlcOutputs.ST30_ET200SP_CM_4xIO_Link_2[21];
	HwOutputs.ST30_ET200SP_CM_4xIO_Link_2[22] := PlcOutputs.ST30_ET200SP_CM_4xIO_Link_2[22];
	HwOutputs.ST30_ET200SP_CM_4xIO_Link_2[23] := PlcOutputs.ST30_ET200SP_CM_4xIO_Link_2[23];
	HwOutputs.ST30_ET200SP_CM_4xIO_Link_2[24] := PlcOutputs.ST30_ET200SP_CM_4xIO_Link_2[24];
	HwOutputs.ST30_ET200SP_CM_4xIO_Link_2[25] := PlcOutputs.ST30_ET200SP_CM_4xIO_Link_2[25];
	HwOutputs.ST30_ET200SP_CM_4xIO_Link_2[26] := PlcOutputs.ST30_ET200SP_CM_4xIO_Link_2[26];
	HwOutputs.ST30_ET200SP_CM_4xIO_Link_2[27] := PlcOutputs.ST30_ET200SP_CM_4xIO_Link_2[27];
	HwOutputs.ST30_ET200SP_CM_4xIO_Link_2[28] := PlcOutputs.ST30_ET200SP_CM_4xIO_Link_2[28];
	HwOutputs.ST30_ET200SP_CM_4xIO_Link_2[29] := PlcOutputs.ST30_ET200SP_CM_4xIO_Link_2[29];
	HwOutputs.ST30_ET200SP_CM_4xIO_Link_2[30] := PlcOutputs.ST30_ET200SP_CM_4xIO_Link_2[30];
	HwOutputs.ST30_ET200SP_CM_4xIO_Link_2[31] := PlcOutputs.ST30_ET200SP_CM_4xIO_Link_2[31];
	HwOutputs.ST30_ET200SP_DQ_16x24VDC_0_5A_ST_1 := PlcOutputs.ST30_ET200SP_DQ_16x24VDC_0_5A_ST_1;
	HwOutputs.ST30_ET200SP_DQ_16x24VDC_0_5A_ST_2 := PlcOutputs.ST30_ET200SP_DQ_16x24VDC_0_5A_ST_2;
	HwOutputs.ST30_ET200SP_DQ_16x24VDC_0_5A_ST_3 := PlcOutputs.ST30_ET200SP_DQ_16x24VDC_0_5A_ST_3;
	HwOutputs.ST30_ET200SP_DQ_16x24VDC_0_5A_ST_4 := PlcOutputs.ST30_ET200SP_DQ_16x24VDC_0_5A_ST_4;
	HwOutputs.ST30_CPX_MPA1S_VMPA1_FB_EMS_8_8DO_1 := PlcOutputs.ST30_CPX_MPA1S_VMPA1_FB_EMS_8_8DO_1;
	HwOutputs.ST30_CPX_MPA1G_VMPA1_FB_EMG_8_8DO_1 := PlcOutputs.ST30_CPX_MPA1G_VMPA1_FB_EMG_8_8DO_1;
	HwOutputs.ST30_CPX_MPA1G_VMPA1_FB_EMG_8_8DO_2 := PlcOutputs.ST30_CPX_MPA1G_VMPA1_FB_EMG_8_8DO_2;
	HwOutputs.ST30_1_DM260_Acquisition_Control_1 := PlcOutputs.ST30_1_DM260_Acquisition_Control_1;
	HwOutputs.ST30_1_DM260_Results_Control_1 := PlcOutputs.ST30_1_DM260_Results_Control_1;
	HwOutputs.ST30_1_DM260_Soft_Event_Control_1 := PlcOutputs.ST30_1_DM260_Soft_Event_Control_1;
	HwOutputs.ST30_1_DM260_User_Data_64_bytes_1[0] := PlcOutputs.ST30_1_DM260_User_Data_64_bytes_1[0];
	HwOutputs.ST30_1_DM260_User_Data_64_bytes_1[1] := PlcOutputs.ST30_1_DM260_User_Data_64_bytes_1[1];
	HwOutputs.ST30_1_DM260_User_Data_64_bytes_1[2] := PlcOutputs.ST30_1_DM260_User_Data_64_bytes_1[2];
	HwOutputs.ST30_1_DM260_User_Data_64_bytes_1[3] := PlcOutputs.ST30_1_DM260_User_Data_64_bytes_1[3];
	HwOutputs.ST30_1_DM260_User_Data_64_bytes_1[4] := PlcOutputs.ST30_1_DM260_User_Data_64_bytes_1[4];
	HwOutputs.ST30_1_DM260_User_Data_64_bytes_1[5] := PlcOutputs.ST30_1_DM260_User_Data_64_bytes_1[5];
	HwOutputs.ST30_1_DM260_User_Data_64_bytes_1[6] := PlcOutputs.ST30_1_DM260_User_Data_64_bytes_1[6];
	HwOutputs.ST30_1_DM260_User_Data_64_bytes_1[7] := PlcOutputs.ST30_1_DM260_User_Data_64_bytes_1[7];
	HwOutputs.ST30_1_DM260_User_Data_64_bytes_1[8] := PlcOutputs.ST30_1_DM260_User_Data_64_bytes_1[8];
	HwOutputs.ST30_1_DM260_User_Data_64_bytes_1[9] := PlcOutputs.ST30_1_DM260_User_Data_64_bytes_1[9];
	HwOutputs.ST30_1_DM260_User_Data_64_bytes_1[10] := PlcOutputs.ST30_1_DM260_User_Data_64_bytes_1[10];
	HwOutputs.ST30_1_DM260_User_Data_64_bytes_1[11] := PlcOutputs.ST30_1_DM260_User_Data_64_bytes_1[11];
	HwOutputs.ST30_1_DM260_User_Data_64_bytes_1[12] := PlcOutputs.ST30_1_DM260_User_Data_64_bytes_1[12];
	HwOutputs.ST30_1_DM260_User_Data_64_bytes_1[13] := PlcOutputs.ST30_1_DM260_User_Data_64_bytes_1[13];
	HwOutputs.ST30_1_DM260_User_Data_64_bytes_1[14] := PlcOutputs.ST30_1_DM260_User_Data_64_bytes_1[14];
	HwOutputs.ST30_1_DM260_User_Data_64_bytes_1[15] := PlcOutputs.ST30_1_DM260_User_Data_64_bytes_1[15];
	HwOutputs.ST30_1_DM260_User_Data_64_bytes_1[16] := PlcOutputs.ST30_1_DM260_User_Data_64_bytes_1[16];
	HwOutputs.ST30_1_DM260_User_Data_64_bytes_1[17] := PlcOutputs.ST30_1_DM260_User_Data_64_bytes_1[17];
	HwOutputs.ST30_1_DM260_User_Data_64_bytes_1[18] := PlcOutputs.ST30_1_DM260_User_Data_64_bytes_1[18];
	HwOutputs.ST30_1_DM260_User_Data_64_bytes_1[19] := PlcOutputs.ST30_1_DM260_User_Data_64_bytes_1[19];
	HwOutputs.ST30_1_DM260_User_Data_64_bytes_1[20] := PlcOutputs.ST30_1_DM260_User_Data_64_bytes_1[20];
	HwOutputs.ST30_1_DM260_User_Data_64_bytes_1[21] := PlcOutputs.ST30_1_DM260_User_Data_64_bytes_1[21];
	HwOutputs.ST30_1_DM260_User_Data_64_bytes_1[22] := PlcOutputs.ST30_1_DM260_User_Data_64_bytes_1[22];
	HwOutputs.ST30_1_DM260_User_Data_64_bytes_1[23] := PlcOutputs.ST30_1_DM260_User_Data_64_bytes_1[23];
	HwOutputs.ST30_1_DM260_User_Data_64_bytes_1[24] := PlcOutputs.ST30_1_DM260_User_Data_64_bytes_1[24];
	HwOutputs.ST30_1_DM260_User_Data_64_bytes_1[25] := PlcOutputs.ST30_1_DM260_User_Data_64_bytes_1[25];
	HwOutputs.ST30_1_DM260_User_Data_64_bytes_1[26] := PlcOutputs.ST30_1_DM260_User_Data_64_bytes_1[26];
	HwOutputs.ST30_1_DM260_User_Data_64_bytes_1[27] := PlcOutputs.ST30_1_DM260_User_Data_64_bytes_1[27];
	HwOutputs.ST30_1_DM260_User_Data_64_bytes_1[28] := PlcOutputs.ST30_1_DM260_User_Data_64_bytes_1[28];
	HwOutputs.ST30_1_DM260_User_Data_64_bytes_1[29] := PlcOutputs.ST30_1_DM260_User_Data_64_bytes_1[29];
	HwOutputs.ST30_1_DM260_User_Data_64_bytes_1[30] := PlcOutputs.ST30_1_DM260_User_Data_64_bytes_1[30];
	HwOutputs.ST30_1_DM260_User_Data_64_bytes_1[31] := PlcOutputs.ST30_1_DM260_User_Data_64_bytes_1[31];
	HwOutputs.ST30_1_DM260_User_Data_64_bytes_1[32] := PlcOutputs.ST30_1_DM260_User_Data_64_bytes_1[32];
	HwOutputs.ST30_1_DM260_User_Data_64_bytes_1[33] := PlcOutputs.ST30_1_DM260_User_Data_64_bytes_1[33];
	HwOutputs.ST30_1_DM260_User_Data_64_bytes_1[34] := PlcOutputs.ST30_1_DM260_User_Data_64_bytes_1[34];
	HwOutputs.ST30_1_DM260_User_Data_64_bytes_1[35] := PlcOutputs.ST30_1_DM260_User_Data_64_bytes_1[35];
	HwOutputs.ST30_1_DM260_User_Data_64_bytes_1[36] := PlcOutputs.ST30_1_DM260_User_Data_64_bytes_1[36];
	HwOutputs.ST30_1_DM260_User_Data_64_bytes_1[37] := PlcOutputs.ST30_1_DM260_User_Data_64_bytes_1[37];
	HwOutputs.ST30_1_DM260_User_Data_64_bytes_1[38] := PlcOutputs.ST30_1_DM260_User_Data_64_bytes_1[38];
	HwOutputs.ST30_1_DM260_User_Data_64_bytes_1[39] := PlcOutputs.ST30_1_DM260_User_Data_64_bytes_1[39];
	HwOutputs.ST30_1_DM260_User_Data_64_bytes_1[40] := PlcOutputs.ST30_1_DM260_User_Data_64_bytes_1[40];
	HwOutputs.ST30_1_DM260_User_Data_64_bytes_1[41] := PlcOutputs.ST30_1_DM260_User_Data_64_bytes_1[41];
	HwOutputs.ST30_1_DM260_User_Data_64_bytes_1[42] := PlcOutputs.ST30_1_DM260_User_Data_64_bytes_1[42];
	HwOutputs.ST30_1_DM260_User_Data_64_bytes_1[43] := PlcOutputs.ST30_1_DM260_User_Data_64_bytes_1[43];
	HwOutputs.ST30_1_DM260_User_Data_64_bytes_1[44] := PlcOutputs.ST30_1_DM260_User_Data_64_bytes_1[44];
	HwOutputs.ST30_1_DM260_User_Data_64_bytes_1[45] := PlcOutputs.ST30_1_DM260_User_Data_64_bytes_1[45];
	HwOutputs.ST30_1_DM260_User_Data_64_bytes_1[46] := PlcOutputs.ST30_1_DM260_User_Data_64_bytes_1[46];
	HwOutputs.ST30_1_DM260_User_Data_64_bytes_1[47] := PlcOutputs.ST30_1_DM260_User_Data_64_bytes_1[47];
	HwOutputs.ST30_1_DM260_User_Data_64_bytes_1[48] := PlcOutputs.ST30_1_DM260_User_Data_64_bytes_1[48];
	HwOutputs.ST30_1_DM260_User_Data_64_bytes_1[49] := PlcOutputs.ST30_1_DM260_User_Data_64_bytes_1[49];
	HwOutputs.ST30_1_DM260_User_Data_64_bytes_1[50] := PlcOutputs.ST30_1_DM260_User_Data_64_bytes_1[50];
	HwOutputs.ST30_1_DM260_User_Data_64_bytes_1[51] := PlcOutputs.ST30_1_DM260_User_Data_64_bytes_1[51];
	HwOutputs.ST30_1_DM260_User_Data_64_bytes_1[52] := PlcOutputs.ST30_1_DM260_User_Data_64_bytes_1[52];
	HwOutputs.ST30_1_DM260_User_Data_64_bytes_1[53] := PlcOutputs.ST30_1_DM260_User_Data_64_bytes_1[53];
	HwOutputs.ST30_1_DM260_User_Data_64_bytes_1[54] := PlcOutputs.ST30_1_DM260_User_Data_64_bytes_1[54];
	HwOutputs.ST30_1_DM260_User_Data_64_bytes_1[55] := PlcOutputs.ST30_1_DM260_User_Data_64_bytes_1[55];
	HwOutputs.ST30_1_DM260_User_Data_64_bytes_1[56] := PlcOutputs.ST30_1_DM260_User_Data_64_bytes_1[56];
	HwOutputs.ST30_1_DM260_User_Data_64_bytes_1[57] := PlcOutputs.ST30_1_DM260_User_Data_64_bytes_1[57];
	HwOutputs.ST30_1_DM260_User_Data_64_bytes_1[58] := PlcOutputs.ST30_1_DM260_User_Data_64_bytes_1[58];
	HwOutputs.ST30_1_DM260_User_Data_64_bytes_1[59] := PlcOutputs.ST30_1_DM260_User_Data_64_bytes_1[59];
	HwOutputs.ST30_1_DM260_User_Data_64_bytes_1[60] := PlcOutputs.ST30_1_DM260_User_Data_64_bytes_1[60];
	HwOutputs.ST30_1_DM260_User_Data_64_bytes_1[61] := PlcOutputs.ST30_1_DM260_User_Data_64_bytes_1[61];
	HwOutputs.ST30_1_DM260_User_Data_64_bytes_1[62] := PlcOutputs.ST30_1_DM260_User_Data_64_bytes_1[62];
	HwOutputs.ST30_1_DM260_User_Data_64_bytes_1[63] := PlcOutputs.ST30_1_DM260_User_Data_64_bytes_1[63];
	HwOutputs.ST30_1_DM260_User_Data_64_bytes_1[64] := PlcOutputs.ST30_1_DM260_User_Data_64_bytes_1[64];
	HwOutputs.ST30_1_DM260_User_Data_64_bytes_1[65] := PlcOutputs.ST30_1_DM260_User_Data_64_bytes_1[65];
	HwOutputs.ST30_1_DM260_User_Data_64_bytes_1[66] := PlcOutputs.ST30_1_DM260_User_Data_64_bytes_1[66];
	HwOutputs.ST30_1_DM260_User_Data_64_bytes_1[67] := PlcOutputs.ST30_1_DM260_User_Data_64_bytes_1[67];
	HwOutputs.ST30_2_DM260_Acquisition_Control_1 := PlcOutputs.ST30_2_DM260_Acquisition_Control_1;
	HwOutputs.ST30_2_DM260_Results_Control_1 := PlcOutputs.ST30_2_DM260_Results_Control_1;
	HwOutputs.ST30_2_DM260_Soft_Event_Control_1 := PlcOutputs.ST30_2_DM260_Soft_Event_Control_1;
	HwOutputs.ST30_2_DM260_User_Data_64_bytes_1[0] := PlcOutputs.ST30_2_DM260_User_Data_64_bytes_1[0];
	HwOutputs.ST30_2_DM260_User_Data_64_bytes_1[1] := PlcOutputs.ST30_2_DM260_User_Data_64_bytes_1[1];
	HwOutputs.ST30_2_DM260_User_Data_64_bytes_1[2] := PlcOutputs.ST30_2_DM260_User_Data_64_bytes_1[2];
	HwOutputs.ST30_2_DM260_User_Data_64_bytes_1[3] := PlcOutputs.ST30_2_DM260_User_Data_64_bytes_1[3];
	HwOutputs.ST30_2_DM260_User_Data_64_bytes_1[4] := PlcOutputs.ST30_2_DM260_User_Data_64_bytes_1[4];
	HwOutputs.ST30_2_DM260_User_Data_64_bytes_1[5] := PlcOutputs.ST30_2_DM260_User_Data_64_bytes_1[5];
	HwOutputs.ST30_2_DM260_User_Data_64_bytes_1[6] := PlcOutputs.ST30_2_DM260_User_Data_64_bytes_1[6];
	HwOutputs.ST30_2_DM260_User_Data_64_bytes_1[7] := PlcOutputs.ST30_2_DM260_User_Data_64_bytes_1[7];
	HwOutputs.ST30_2_DM260_User_Data_64_bytes_1[8] := PlcOutputs.ST30_2_DM260_User_Data_64_bytes_1[8];
	HwOutputs.ST30_2_DM260_User_Data_64_bytes_1[9] := PlcOutputs.ST30_2_DM260_User_Data_64_bytes_1[9];
	HwOutputs.ST30_2_DM260_User_Data_64_bytes_1[10] := PlcOutputs.ST30_2_DM260_User_Data_64_bytes_1[10];
	HwOutputs.ST30_2_DM260_User_Data_64_bytes_1[11] := PlcOutputs.ST30_2_DM260_User_Data_64_bytes_1[11];
	HwOutputs.ST30_2_DM260_User_Data_64_bytes_1[12] := PlcOutputs.ST30_2_DM260_User_Data_64_bytes_1[12];
	HwOutputs.ST30_2_DM260_User_Data_64_bytes_1[13] := PlcOutputs.ST30_2_DM260_User_Data_64_bytes_1[13];
	HwOutputs.ST30_2_DM260_User_Data_64_bytes_1[14] := PlcOutputs.ST30_2_DM260_User_Data_64_bytes_1[14];
	HwOutputs.ST30_2_DM260_User_Data_64_bytes_1[15] := PlcOutputs.ST30_2_DM260_User_Data_64_bytes_1[15];
	HwOutputs.ST30_2_DM260_User_Data_64_bytes_1[16] := PlcOutputs.ST30_2_DM260_User_Data_64_bytes_1[16];
	HwOutputs.ST30_2_DM260_User_Data_64_bytes_1[17] := PlcOutputs.ST30_2_DM260_User_Data_64_bytes_1[17];
	HwOutputs.ST30_2_DM260_User_Data_64_bytes_1[18] := PlcOutputs.ST30_2_DM260_User_Data_64_bytes_1[18];
	HwOutputs.ST30_2_DM260_User_Data_64_bytes_1[19] := PlcOutputs.ST30_2_DM260_User_Data_64_bytes_1[19];
	HwOutputs.ST30_2_DM260_User_Data_64_bytes_1[20] := PlcOutputs.ST30_2_DM260_User_Data_64_bytes_1[20];
	HwOutputs.ST30_2_DM260_User_Data_64_bytes_1[21] := PlcOutputs.ST30_2_DM260_User_Data_64_bytes_1[21];
	HwOutputs.ST30_2_DM260_User_Data_64_bytes_1[22] := PlcOutputs.ST30_2_DM260_User_Data_64_bytes_1[22];
	HwOutputs.ST30_2_DM260_User_Data_64_bytes_1[23] := PlcOutputs.ST30_2_DM260_User_Data_64_bytes_1[23];
	HwOutputs.ST30_2_DM260_User_Data_64_bytes_1[24] := PlcOutputs.ST30_2_DM260_User_Data_64_bytes_1[24];
	HwOutputs.ST30_2_DM260_User_Data_64_bytes_1[25] := PlcOutputs.ST30_2_DM260_User_Data_64_bytes_1[25];
	HwOutputs.ST30_2_DM260_User_Data_64_bytes_1[26] := PlcOutputs.ST30_2_DM260_User_Data_64_bytes_1[26];
	HwOutputs.ST30_2_DM260_User_Data_64_bytes_1[27] := PlcOutputs.ST30_2_DM260_User_Data_64_bytes_1[27];
	HwOutputs.ST30_2_DM260_User_Data_64_bytes_1[28] := PlcOutputs.ST30_2_DM260_User_Data_64_bytes_1[28];
	HwOutputs.ST30_2_DM260_User_Data_64_bytes_1[29] := PlcOutputs.ST30_2_DM260_User_Data_64_bytes_1[29];
	HwOutputs.ST30_2_DM260_User_Data_64_bytes_1[30] := PlcOutputs.ST30_2_DM260_User_Data_64_bytes_1[30];
	HwOutputs.ST30_2_DM260_User_Data_64_bytes_1[31] := PlcOutputs.ST30_2_DM260_User_Data_64_bytes_1[31];
	HwOutputs.ST30_2_DM260_User_Data_64_bytes_1[32] := PlcOutputs.ST30_2_DM260_User_Data_64_bytes_1[32];
	HwOutputs.ST30_2_DM260_User_Data_64_bytes_1[33] := PlcOutputs.ST30_2_DM260_User_Data_64_bytes_1[33];
	HwOutputs.ST30_2_DM260_User_Data_64_bytes_1[34] := PlcOutputs.ST30_2_DM260_User_Data_64_bytes_1[34];
	HwOutputs.ST30_2_DM260_User_Data_64_bytes_1[35] := PlcOutputs.ST30_2_DM260_User_Data_64_bytes_1[35];
	HwOutputs.ST30_2_DM260_User_Data_64_bytes_1[36] := PlcOutputs.ST30_2_DM260_User_Data_64_bytes_1[36];
	HwOutputs.ST30_2_DM260_User_Data_64_bytes_1[37] := PlcOutputs.ST30_2_DM260_User_Data_64_bytes_1[37];
	HwOutputs.ST30_2_DM260_User_Data_64_bytes_1[38] := PlcOutputs.ST30_2_DM260_User_Data_64_bytes_1[38];
	HwOutputs.ST30_2_DM260_User_Data_64_bytes_1[39] := PlcOutputs.ST30_2_DM260_User_Data_64_bytes_1[39];
	HwOutputs.ST30_2_DM260_User_Data_64_bytes_1[40] := PlcOutputs.ST30_2_DM260_User_Data_64_bytes_1[40];
	HwOutputs.ST30_2_DM260_User_Data_64_bytes_1[41] := PlcOutputs.ST30_2_DM260_User_Data_64_bytes_1[41];
	HwOutputs.ST30_2_DM260_User_Data_64_bytes_1[42] := PlcOutputs.ST30_2_DM260_User_Data_64_bytes_1[42];
	HwOutputs.ST30_2_DM260_User_Data_64_bytes_1[43] := PlcOutputs.ST30_2_DM260_User_Data_64_bytes_1[43];
	HwOutputs.ST30_2_DM260_User_Data_64_bytes_1[44] := PlcOutputs.ST30_2_DM260_User_Data_64_bytes_1[44];
	HwOutputs.ST30_2_DM260_User_Data_64_bytes_1[45] := PlcOutputs.ST30_2_DM260_User_Data_64_bytes_1[45];
	HwOutputs.ST30_2_DM260_User_Data_64_bytes_1[46] := PlcOutputs.ST30_2_DM260_User_Data_64_bytes_1[46];
	HwOutputs.ST30_2_DM260_User_Data_64_bytes_1[47] := PlcOutputs.ST30_2_DM260_User_Data_64_bytes_1[47];
	HwOutputs.ST30_2_DM260_User_Data_64_bytes_1[48] := PlcOutputs.ST30_2_DM260_User_Data_64_bytes_1[48];
	HwOutputs.ST30_2_DM260_User_Data_64_bytes_1[49] := PlcOutputs.ST30_2_DM260_User_Data_64_bytes_1[49];
	HwOutputs.ST30_2_DM260_User_Data_64_bytes_1[50] := PlcOutputs.ST30_2_DM260_User_Data_64_bytes_1[50];
	HwOutputs.ST30_2_DM260_User_Data_64_bytes_1[51] := PlcOutputs.ST30_2_DM260_User_Data_64_bytes_1[51];
	HwOutputs.ST30_2_DM260_User_Data_64_bytes_1[52] := PlcOutputs.ST30_2_DM260_User_Data_64_bytes_1[52];
	HwOutputs.ST30_2_DM260_User_Data_64_bytes_1[53] := PlcOutputs.ST30_2_DM260_User_Data_64_bytes_1[53];
	HwOutputs.ST30_2_DM260_User_Data_64_bytes_1[54] := PlcOutputs.ST30_2_DM260_User_Data_64_bytes_1[54];
	HwOutputs.ST30_2_DM260_User_Data_64_bytes_1[55] := PlcOutputs.ST30_2_DM260_User_Data_64_bytes_1[55];
	HwOutputs.ST30_2_DM260_User_Data_64_bytes_1[56] := PlcOutputs.ST30_2_DM260_User_Data_64_bytes_1[56];
	HwOutputs.ST30_2_DM260_User_Data_64_bytes_1[57] := PlcOutputs.ST30_2_DM260_User_Data_64_bytes_1[57];
	HwOutputs.ST30_2_DM260_User_Data_64_bytes_1[58] := PlcOutputs.ST30_2_DM260_User_Data_64_bytes_1[58];
	HwOutputs.ST30_2_DM260_User_Data_64_bytes_1[59] := PlcOutputs.ST30_2_DM260_User_Data_64_bytes_1[59];
	HwOutputs.ST30_2_DM260_User_Data_64_bytes_1[60] := PlcOutputs.ST30_2_DM260_User_Data_64_bytes_1[60];
	HwOutputs.ST30_2_DM260_User_Data_64_bytes_1[61] := PlcOutputs.ST30_2_DM260_User_Data_64_bytes_1[61];
	HwOutputs.ST30_2_DM260_User_Data_64_bytes_1[62] := PlcOutputs.ST30_2_DM260_User_Data_64_bytes_1[62];
	HwOutputs.ST30_2_DM260_User_Data_64_bytes_1[63] := PlcOutputs.ST30_2_DM260_User_Data_64_bytes_1[63];
	HwOutputs.ST30_2_DM260_User_Data_64_bytes_1[64] := PlcOutputs.ST30_2_DM260_User_Data_64_bytes_1[64];
	HwOutputs.ST30_2_DM260_User_Data_64_bytes_1[65] := PlcOutputs.ST30_2_DM260_User_Data_64_bytes_1[65];
	HwOutputs.ST30_2_DM260_User_Data_64_bytes_1[66] := PlcOutputs.ST30_2_DM260_User_Data_64_bytes_1[66];
	HwOutputs.ST30_2_DM260_User_Data_64_bytes_1[67] := PlcOutputs.ST30_2_DM260_User_Data_64_bytes_1[67];
END_FUNCTION
